FUNCTION_BLOCK CarLightCtl_Discrete (* Function block for controling the operation of a car trafic light following the rules of Germany *)
  (* Standard: 61499-2 *)
  (* Version 0.0, 2014-07-11, 4DIAC-IDE, 4DIAC-Consortium *)
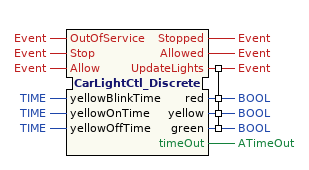
  EVENT_INPUT
    OutOfService;
    Stop;
    Allow;
  END_EVENT
  EVENT_OUTPUT
    Stopped;
    Allowed;
    UpdateLights WITH green, red, yellow;
  END_EVENT
  VAR_INPUT
    yellowBlinkTime : TIME; (* Cycle time for the yellow light blinking in out of service *)
    yellowOnTime : TIME; (* Time the yellow light is on when switching from red to green *)
    yellowOffTime : TIME; (* Time the yellow light is on when swithcing from green to red *)
  END_VAR
  VAR_OUTPUT
    red : BOOL;
    yellow : BOOL;
    green : BOOL;
  END_VAR
  PLUGS
    timeOut : ATimeOut;
  END_PLUGS
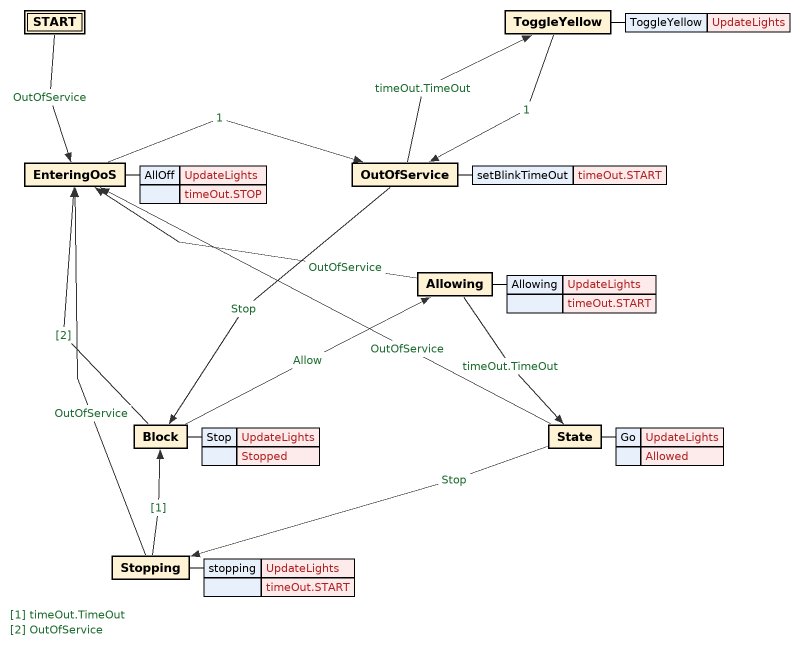
  EC_STATES
    START;
    OutOfService : setBlinkTimeOut -> timeOut.START;
    Block : Stop -> UpdateLights, -> Stopped;
    State : Go -> UpdateLights, -> Allowed;
    ToggleYellow : ToggleYellow -> UpdateLights;
    EnteringOoS : AllOff -> UpdateLights, -> timeOut.STOP;
    Allowing : Allowing -> UpdateLights, -> timeOut.START;
    Stopping : stopping -> UpdateLights, -> timeOut.START;
  END_STATES
  EC_TRANSITIONS
    OutOfService TO Block := Stop;
    OutOfService TO ToggleYellow := timeOut.TimeOut;
    ToggleYellow TO OutOfService := 1;
    START TO EnteringOoS := OutOfService;
    Block TO EnteringOoS := OutOfService;
    State TO EnteringOoS := OutOfService;
    EnteringOoS TO OutOfService := 1;
    Block TO Allowing := Allow;
    Allowing TO State := timeOut.TimeOut;
    State TO Stopping := Stop;
    Stopping TO EnteringOoS := OutOfService;
    Stopping TO Block := timeOut.TimeOut;
    Allowing TO EnteringOoS := OutOfService;
  END_TRANSITIONS
  ALGORITHM AllOff IN ST:
red := FALSE;
yellow := FALSE;
green := FALSE;
  END_ALGORITHM
  ALGORITHM Stop IN ST: (* Put lights in stop mode (i.e., red := true, green := false) *)
red := TRUE;
yellow := FALSE;
green := FALSE;
  END_ALGORITHM
  ALGORITHM Go IN ST: (* Put lights in Walk mode (i.e., red := false, green := true) *)
red := FALSE;
yellow := FALSE;
green := TRUE;
  END_ALGORITHM
  ALGORITHM setBlinkTimeOut IN ST:
timeOut.DT := yellowBlinkTime;
  END_ALGORITHM
  ALGORITHM ToggleYellow IN ST: (* new algorithm *)
yellow := NOT yellow;
  END_ALGORITHM
  ALGORITHM Allowing IN ST: (* new algorithm *)
yellow := TRUE;
timeOut.DT := yellowOnTime;
  END_ALGORITHM
  ALGORITHM stopping IN ST: (* new algorithm *)
green := FALSE;
yellow := TRUE;

timeOut.DT := yellowOffTime;
  END_ALGORITHM
END_FUNCTION_BLOCK
